FUNCTION TijdVanWakkerWorden : BOOL
VAR_INPUT
    ActueleUur   : INT;
    ActueleMinuut : INT;
    WekUur      : INT;
    WekMinuut    : INT;
END_VAR



IF (ActueleUur = WekUur) AND (ActueleMinuut = Wekminuut) THEN
    TijdVanWakkerWorden := TRUE;
ELSE
    TijdVanWakkerWorden := FALSE;
END_IF

END_FUNCTION

(* stored: Version 1.1.0.1, ProductVersion 3.1.4024.15
   POU Functieprogramma: Id {19053d2d-3e91-4fef-9b84-b5856a8124db}, SpecialFunc None *)
